// TIA Portal V16 export
// export: Created 2024-06-24T15:42:28.1265096Z, ExportSetting WithDefaults, DisplayName Totally Integrated Automation Portal, DisplayVersion V16, DisplayName TIA Portal Version Control Interface, DisplayVersion V16, DisplayName TIA Portal Openness, DisplayVersion V16, DisplayName STEP 7 Professional, DisplayVersion V16, DisplayName STEP 7 Safety, DisplayVersion V16, DisplayName WinCC Advanced, DisplayVersion V16
ORGANIZATION_BLOCK "OB_WeightSorter"   // OB128, LAD, ProgramCycle
TITLE = "Main Program Sweep (Cycle)"
{ S7_Optimized_Access := 'TRUE' }
VERSION : 0.1
// stored: AutoNumber true, IsIECCheckEnabled false, SetENOAutomatically false
   VAR_INPUT
      Initial_Call : Bool;   // Initial call of this OB
      Remanence : Bool;   // =True, if remanent data are available
   END_VAR
   VAR_TEMP   // added for the SCL form of the ladder/FBD networks
      _w1 : Bool;
   END_VAR
BEGIN

REGION Network 1
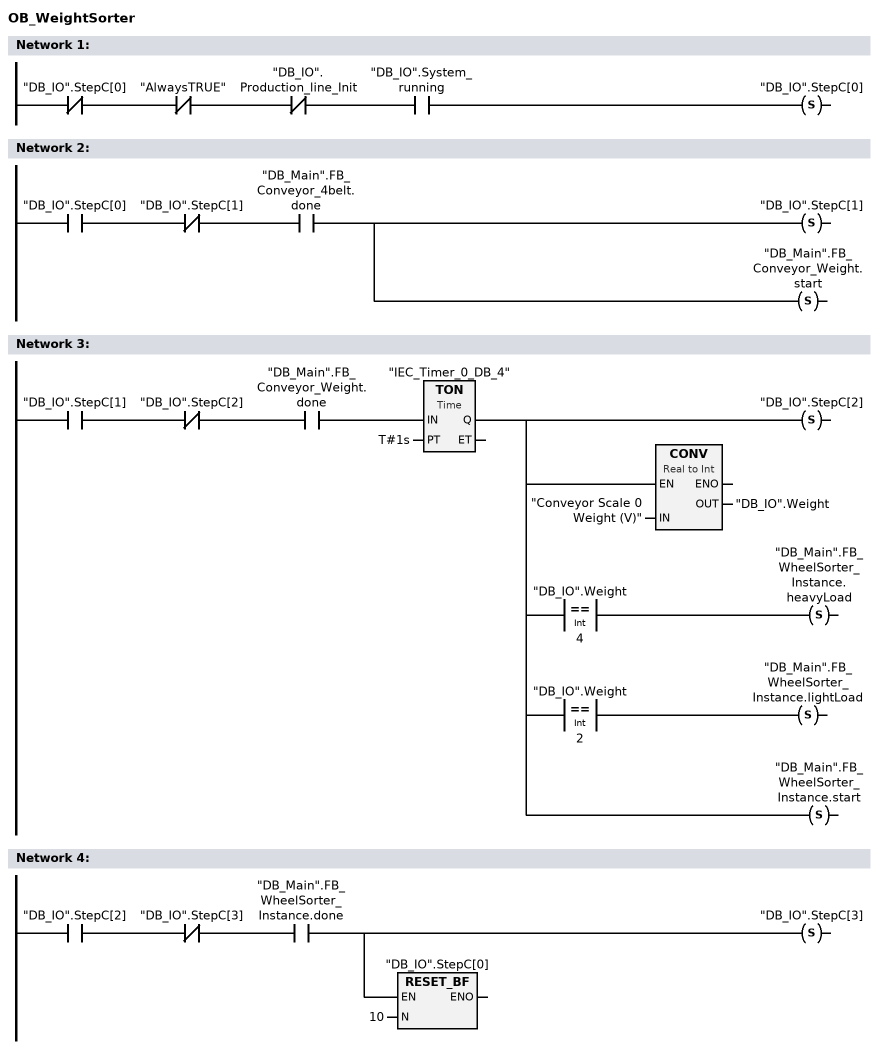
   RUNG wire#powerrail
      I_Contact( "DB_IO".StepC[0] )
      I_Contact( "AlwaysTRUE" )
      I_Contact( "DB_IO".Production_line_Init )
      Contact( "DB_IO".System_running )
      S_Coil( "DB_IO".StepC[0] )
   END_RUNG
   // the same network as SCL:
   IF NOT "DB_IO".StepC[0] AND NOT "AlwaysTRUE" AND NOT "DB_IO".Production_line_Init AND "DB_IO".System_running THEN
       "DB_IO".StepC[0] := TRUE;
   END_IF;
END_REGION

REGION Network 2
   RUNG wire#powerrail
      Contact( "DB_IO".StepC[0] )
      I_Contact( "DB_IO".StepC[1] )
      Contact( "DB_Main".FB_Conveyor_4belt.done )
      wire#w1
      S_Coil( "DB_IO".StepC[1] )
   END_RUNG
   RUNG wire#w1
      S_Coil( "DB_Main".FB_Conveyor_Weight.start )
   END_RUNG
   // the same network as SCL:
   #_w1 := "DB_IO".StepC[0] AND NOT "DB_IO".StepC[1] AND "DB_Main".FB_Conveyor_4belt.done;
   IF #_w1 THEN
       "DB_IO".StepC[1] := TRUE;
       "DB_Main".FB_Conveyor_Weight.start := TRUE;
   END_IF;
END_REGION

REGION Network 3
   RUNG wire#powerrail
      Contact( "DB_IO".StepC[1] )
      I_Contact( "DB_IO".StepC[2] )
      Contact( "DB_Main".FB_Conveyor_Weight.done )
      { S7_Templates := "time_type := Time" } "IEC_Timer_0_DB_4".TON(pt := T#1s, et =>)
      wire#w1
      S_Coil( "DB_IO".StepC[2] )
   END_RUNG
   RUNG wire#w1
      { S7_Templates := "[SrcType := Real, DestType := Int]" } Convert(in := "Conveyor Scale 0 Weight (V)", out => "DB_IO".Weight)
   END_RUNG
   RUNG wire#w1
      { S7_Templates := "SrcType := Int" } EQ_Contact(in1 := "DB_IO".Weight, in2 := 4)
      S_Coil( "DB_Main".FB_WheelSorter_Instance.heavyLoad )
   END_RUNG
   RUNG wire#w1
      { S7_Templates := "SrcType := Int" } EQ_Contact(in1 := "DB_IO".Weight, in2 := 2)
      S_Coil( "DB_Main".FB_WheelSorter_Instance.lightLoad )
   END_RUNG
   RUNG wire#w1
      S_Coil( "DB_Main".FB_WheelSorter_Instance.start )
   END_RUNG
   // the same network as SCL:
   "IEC_Timer_0_DB_4".TON(IN := "DB_IO".StepC[1] AND NOT "DB_IO".StepC[2] AND "DB_Main".FB_Conveyor_Weight.done,
                          PT := T#1s);
   IF "IEC_Timer_0_DB_4".Q THEN
       "DB_IO".StepC[2] := TRUE;
       "DB_IO".Weight := REAL_TO_INT("Conveyor Scale 0 Weight (V)");
   END_IF;
   IF "IEC_Timer_0_DB_4".Q AND ("DB_IO".Weight = 4) THEN
       "DB_Main".FB_WheelSorter_Instance.heavyLoad := TRUE;
   END_IF;
   IF "IEC_Timer_0_DB_4".Q AND ("DB_IO".Weight = 2) THEN
       "DB_Main".FB_WheelSorter_Instance.lightLoad := TRUE;
   END_IF;
   IF "IEC_Timer_0_DB_4".Q THEN "DB_Main".FB_WheelSorter_Instance.start := TRUE; END_IF;
END_REGION

REGION Network 4
   // no SCL statement known for RBitfield: written as a call
   #_w1 := "DB_IO".StepC[2] AND NOT "DB_IO".StepC[3] AND "DB_Main".FB_WheelSorter_Instance.done;
   IF #_w1 THEN
       "DB_IO".StepC[3] := TRUE;
       RESET_BF(operand := "DB_IO".StepC[0], n := 10);
   END_IF;
END_REGION
END_ORGANIZATION_BLOCK
